# EPICS autosave request: iocBoot/sioc-spd-im01/sioc-spd-im01.req
file "lcls2.req" AREA=SPD,POS=695
